# EPICS substitutions: XF_PPSApp/Db/plc-dint-only-b.substitutions
# Data is received from asyn device in arrays of double words (DINTs)
# Parse the element in longin, no macro definition
# Each DINT can have a grouping label for encoded data
file longin-only-b.template {
    pattern { "" }
            { "" }
}
